SUBAPPLICATION mapping (* Subapplication Type *)
  (* Standard: 61499-2 *)
  (* Version 1.0, 2023-02-19, franz *)
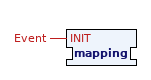
  EVENT_INPUT
    INIT;
  END_EVENT
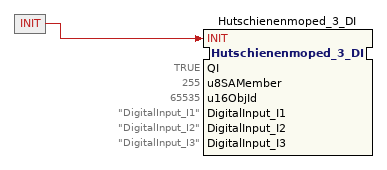
  FBS
    Hutschienenmoped_3_DI : Hutschienenmoped_3_DI(QI := TRUE, u8SAMember := 255, u16ObjId := 65535, DigitalInput_I1 := "DigitalInput_I1", DigitalInput_I2 := "DigitalInput_I2", DigitalInput_I3 := "DigitalInput_I3");
  END_FBS
  EVENT_CONNECTIONS
    INIT TO Hutschienenmoped_3_DI.INIT;
  END_CONNECTIONS
END_SUBAPPLICATION
